Xinje XDPPro project, PLC1: XD5-60-6Pls (software 3.4 2016-10-12)

PROGRAM Ladder

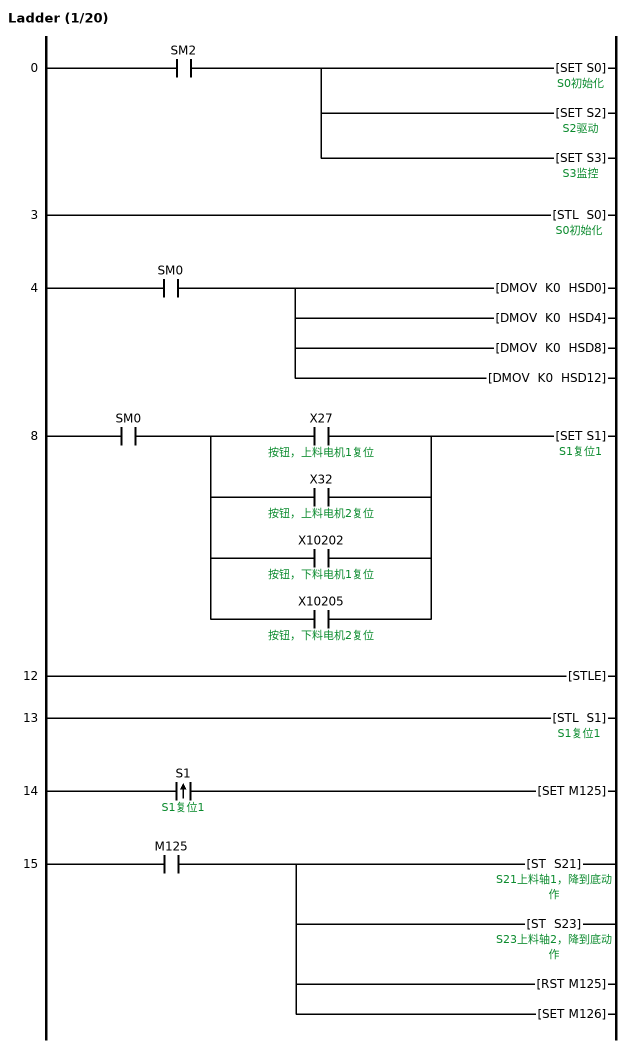
LD     SM2
SET    S0	; S0初始化
SET    S2	; S2驱动
SET    S3	; S3监控
STL    S0	; S0初始化
LD     SM0
DMOV   K0 HSD0
DMOV   K0 HSD4
DMOV   K0 HSD8
DMOV   K0 HSD12
LD     SM0
LD     X27	; 按钮，上料电机1复位
OR     X32	; 按钮，上料电机2复位
OR     X10202	; 按钮，下料电机1复位
OR     X10205	; 按钮，下料电机2复位
ANB
SET    S1	; S1复位1
STLE
STL    S1	; S1复位1
LDP    S1	; S1复位1
SET    M125
LD     M125
ST     S21	; S21上料轴1，降到底动作
ST     S23	; S23上料轴2，降到底动作
RST    M125
SET    M126

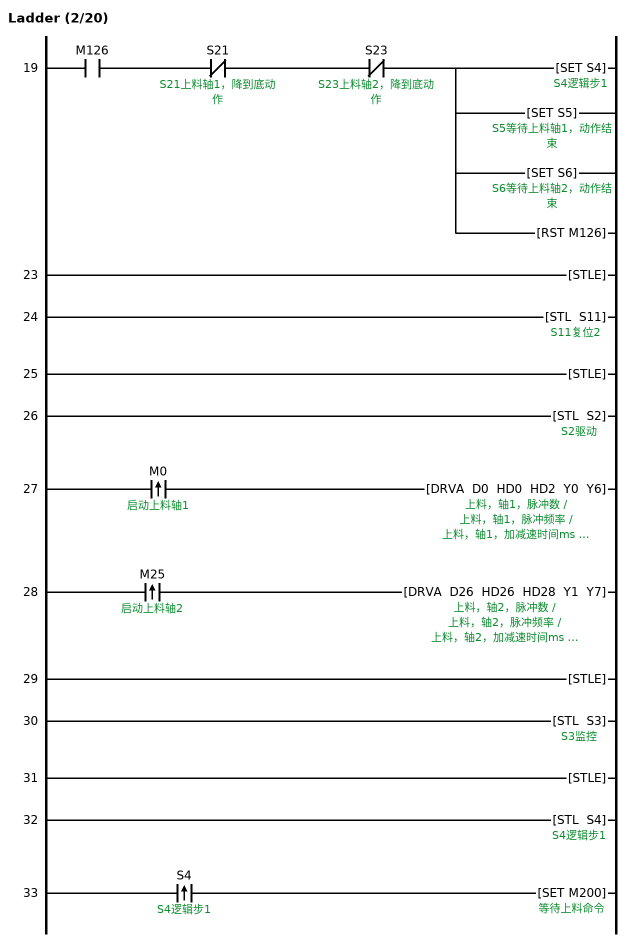
LD     M126
ANI    S21	; S21上料轴1，降到底动作
ANI    S23	; S23上料轴2，降到底动作
SET    S4	; S4逻辑步1
SET    S5	; S5等待上料轴1，动作结束
SET    S6	; S6等待上料轴2，动作结束
RST    M126
STLE
STL    S11	; S11复位2
STLE
STL    S2	; S2驱动
LDP    M0	; 启动上料轴1
DRVA   D0 HD0 HD2 Y0 Y6	; 上料，轴1，脉冲数 / 上料，轴1，脉冲频率 / 上料，轴1，加减速时间ms / 上料1电机脉冲 / 上料1电机方向
LDP    M25	; 启动上料轴2
DRVA   D26 HD26 HD28 Y1 Y7	; 上料，轴2，脉冲数 / 上料，轴2，脉冲频率 / 上料，轴2，加减速时间ms / 上料2电机脉冲 / 上料2电机方向
STLE
STL    S3	; S3监控
STLE
STL    S4	; S4逻辑步1
LDP    S4	; S4逻辑步1
SET    M200	; 等待上料命令

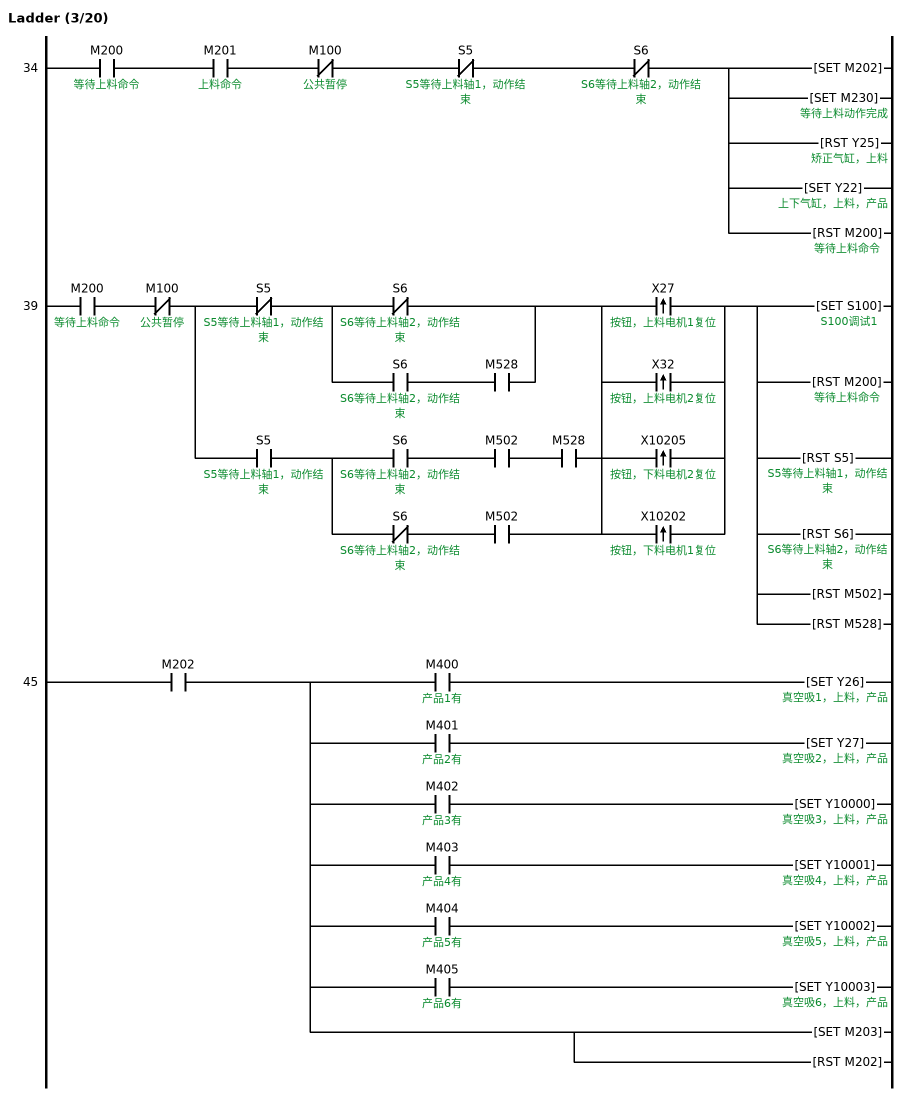
LD     M200	; 等待上料命令
AND    M201	; 上料命令
ANI    M100	; 公共暂停
ANI    S5	; S5等待上料轴1，动作结束
ANI    S6	; S6等待上料轴2，动作结束
SET    M202
SET    M230	; 等待上料动作完成
RST    Y25	; 矫正气缸，上料
SET    Y22	; 上下气缸，上料，产品
RST    M200	; 等待上料命令
LD     M200	; 等待上料命令
ANI    M100	; 公共暂停
LDI    S5	; S5等待上料轴1，动作结束
LDI    S6	; S6等待上料轴2，动作结束
LD     S6	; S6等待上料轴2，动作结束
AND    M528
ORB
ANB
LD     S5	; S5等待上料轴1，动作结束
LD     S6	; S6等待上料轴2，动作结束
AND    M502
AND    M528
LDI    S6	; S6等待上料轴2，动作结束
AND    M502
ORB
ANB
ORB
ANB
LDP    X27	; 按钮，上料电机1复位
ORP    X32	; 按钮，上料电机2复位
ORP    X10205	; 按钮，下料电机2复位
ORP    X10202	; 按钮，下料电机1复位
ANB
SET    S100	; S100调试1
RST    M200	; 等待上料命令
RST    S5	; S5等待上料轴1，动作结束
RST    S6	; S6等待上料轴2，动作结束
RST    M502
RST    M528
LD     M202
MPS
AND    M400	; 产品1有
SET    Y26	; 真空吸1，上料，产品
MRD
AND    M401	; 产品2有
SET    Y27	; 真空吸2，上料，产品
MRD
AND    M402	; 产品3有
SET    Y10000	; 真空吸3，上料，产品
MRD
AND    M403	; 产品4有
SET    Y10001	; 真空吸4，上料，产品
MRD
AND    M404	; 产品5有
SET    Y10002	; 真空吸5，上料，产品
MRD
AND    M405	; 产品6有
SET    Y10003	; 真空吸6，上料，产品
MPP
SET    M203
RST    M202

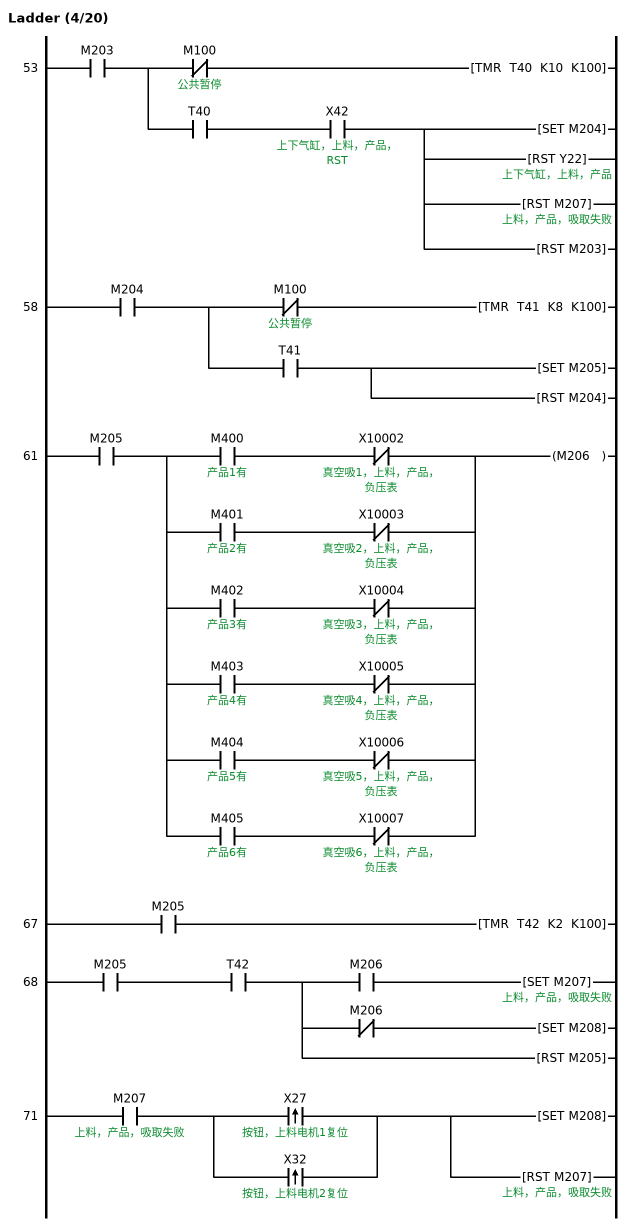
LD     M203
MPS
ANI    M100	; 公共暂停
TMR    T40 K10 K100
MPP
AND    T40
AND    X42	; 上下气缸，上料，产品，RST
SET    M204
RST    Y22	; 上下气缸，上料，产品
RST    M207	; 上料，产品，吸取失败
RST    M203
LD     M204
MPS
ANI    M100	; 公共暂停
TMR    T41 K8 K100
MPP
AND    T41
SET    M205
RST    M204
LD     M205
LD     M400	; 产品1有
ANI    X10002	; 真空吸1，上料，产品，负压表
LD     M401	; 产品2有
ANI    X10003	; 真空吸2，上料，产品，负压表
ORB
LD     M402	; 产品3有
ANI    X10004	; 真空吸3，上料，产品，负压表
ORB
LD     M403	; 产品4有
ANI    X10005	; 真空吸4，上料，产品，负压表
ORB
LD     M404	; 产品5有
ANI    X10006	; 真空吸5，上料，产品，负压表
ORB
LD     M405	; 产品6有
ANI    X10007	; 真空吸6，上料，产品，负压表
ORB
ANB
OUT    M206
LD     M205
TMR    T42 K2 K100
LD     M205
AND    T42
MPS
AND    M206
SET    M207	; 上料，产品，吸取失败
MRD
ANI    M206
SET    M208
MPP
RST    M205
LD     M207	; 上料，产品，吸取失败
LDP    X27	; 按钮，上料电机1复位
ORP    X32	; 按钮，上料电机2复位
ANB
SET    M208
RST    M207	; 上料，产品，吸取失败

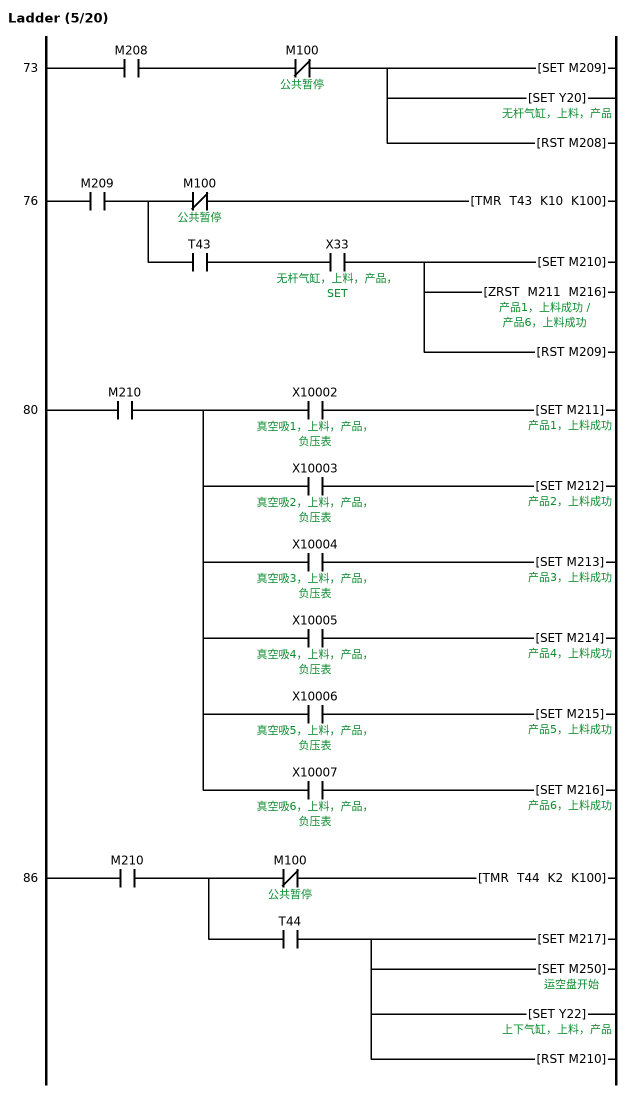
LD     M208
ANI    M100	; 公共暂停
SET    M209
SET    Y20	; 无杆气缸，上料，产品
RST    M208
LD     M209
MPS
ANI    M100	; 公共暂停
TMR    T43 K10 K100
MPP
AND    T43
AND    X33	; 无杆气缸，上料，产品，SET
SET    M210
ZRST   M211 M216	; 产品1，上料成功 / 产品6，上料成功
RST    M209
LD     M210
MPS
AND    X10002	; 真空吸1，上料，产品，负压表
SET    M211	; 产品1，上料成功
MRD
AND    X10003	; 真空吸2，上料，产品，负压表
SET    M212	; 产品2，上料成功
MRD
AND    X10004	; 真空吸3，上料，产品，负压表
SET    M213	; 产品3，上料成功
MRD
AND    X10005	; 真空吸4，上料，产品，负压表
SET    M214	; 产品4，上料成功
MRD
AND    X10006	; 真空吸5，上料，产品，负压表
SET    M215	; 产品5，上料成功
MPP
AND    X10007	; 真空吸6，上料，产品，负压表
SET    M216	; 产品6，上料成功
LD     M210
MPS
ANI    M100	; 公共暂停
TMR    T44 K2 K100
MPP
AND    T44
SET    M217
SET    M250	; 运空盘开始
SET    Y22	; 上下气缸，上料，产品
RST    M210

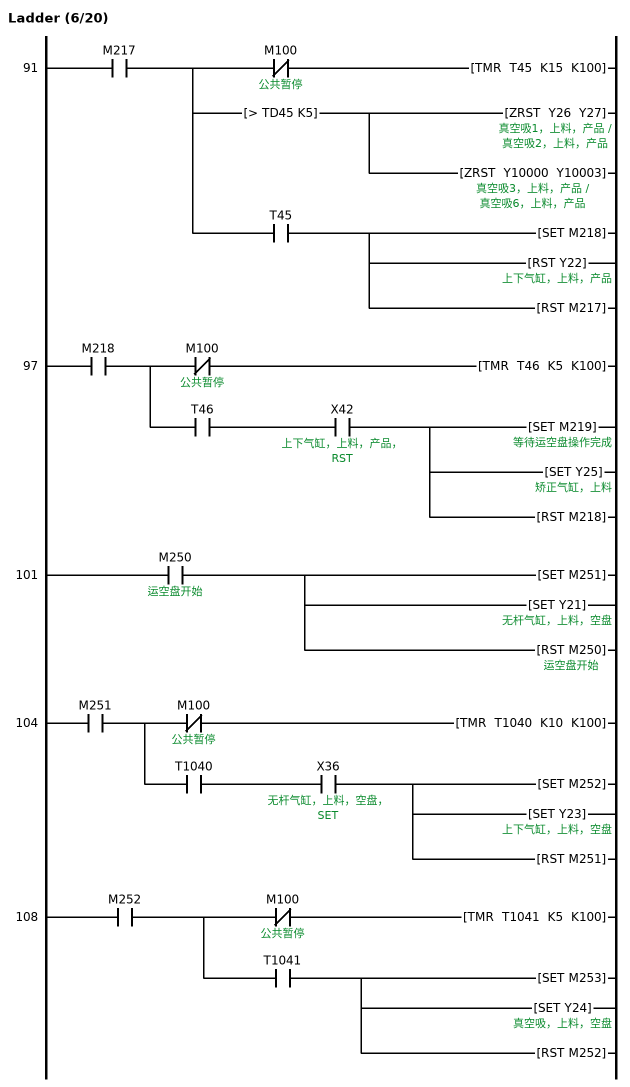
LD     M217
MPS
ANI    M100	; 公共暂停
TMR    T45 K15 K100
MRD
AND>   TD45 K5
ZRST   Y26 Y27	; 真空吸1，上料，产品 / 真空吸2，上料，产品
ZRST   Y10000 Y10003	; 真空吸3，上料，产品 / 真空吸6，上料，产品
MPP
AND    T45
SET    M218
RST    Y22	; 上下气缸，上料，产品
RST    M217
LD     M218
MPS
ANI    M100	; 公共暂停
TMR    T46 K5 K100
MPP
AND    T46
AND    X42	; 上下气缸，上料，产品，RST
SET    M219	; 等待运空盘操作完成
SET    Y25	; 矫正气缸，上料
RST    M218
LD     M250	; 运空盘开始
SET    M251
SET    Y21	; 无杆气缸，上料，空盘
RST    M250	; 运空盘开始
LD     M251
MPS
ANI    M100	; 公共暂停
TMR    T1040 K10 K100
MPP
AND    T1040
AND    X36	; 无杆气缸，上料，空盘，SET
SET    M252
SET    Y23	; 上下气缸，上料，空盘
RST    M251
LD     M252
MPS
ANI    M100	; 公共暂停
TMR    T1041 K5 K100
MPP
AND    T1041
SET    M253
SET    Y24	; 真空吸，上料，空盘
RST    M252

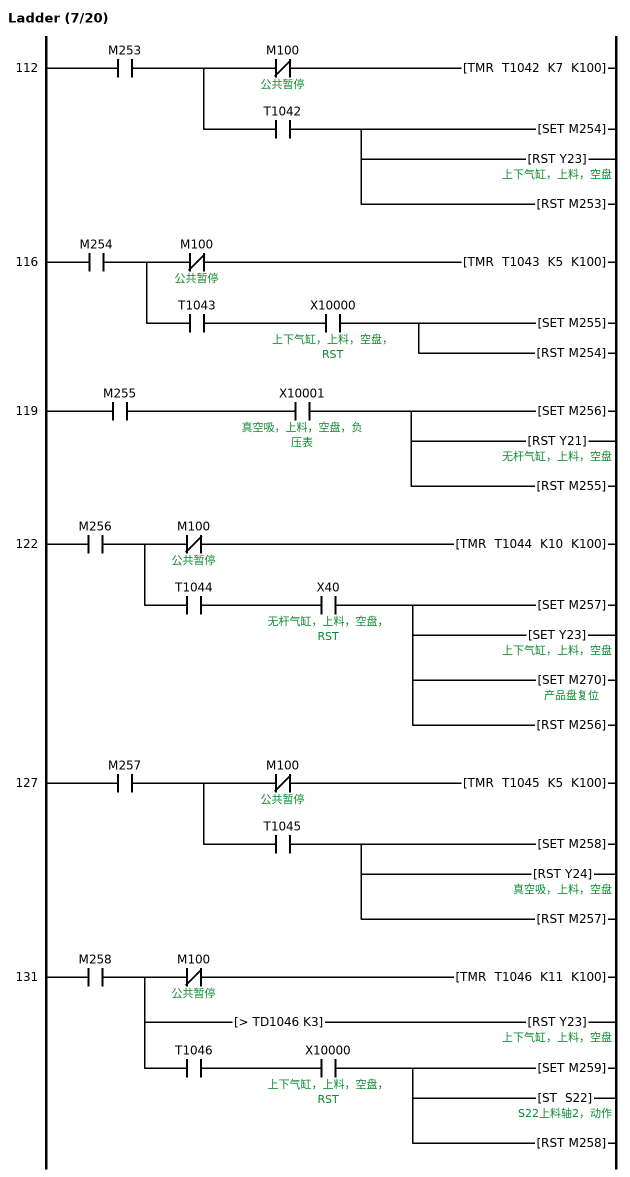
LD     M253
MPS
ANI    M100	; 公共暂停
TMR    T1042 K7 K100
MPP
AND    T1042
SET    M254
RST    Y23	; 上下气缸，上料，空盘
RST    M253
LD     M254
MPS
ANI    M100	; 公共暂停
TMR    T1043 K5 K100
MPP
AND    T1043
AND    X10000	; 上下气缸，上料，空盘，RST
SET    M255
RST    M254
LD     M255
AND    X10001	; 真空吸，上料，空盘，负压表
SET    M256
RST    Y21	; 无杆气缸，上料，空盘
RST    M255
LD     M256
MPS
ANI    M100	; 公共暂停
TMR    T1044 K10 K100
MPP
AND    T1044
AND    X40	; 无杆气缸，上料，空盘，RST
SET    M257
SET    Y23	; 上下气缸，上料，空盘
SET    M270	; 产品盘复位
RST    M256
LD     M257
MPS
ANI    M100	; 公共暂停
TMR    T1045 K5 K100
MPP
AND    T1045
SET    M258
RST    Y24	; 真空吸，上料，空盘
RST    M257
LD     M258
MPS
ANI    M100	; 公共暂停
TMR    T1046 K11 K100
MRD
AND>   TD1046 K3
RST    Y23	; 上下气缸，上料，空盘
MPP
AND    T1046
AND    X10000	; 上下气缸，上料，空盘，RST
SET    M259
ST     S22	; S22上料轴2，动作
RST    M258

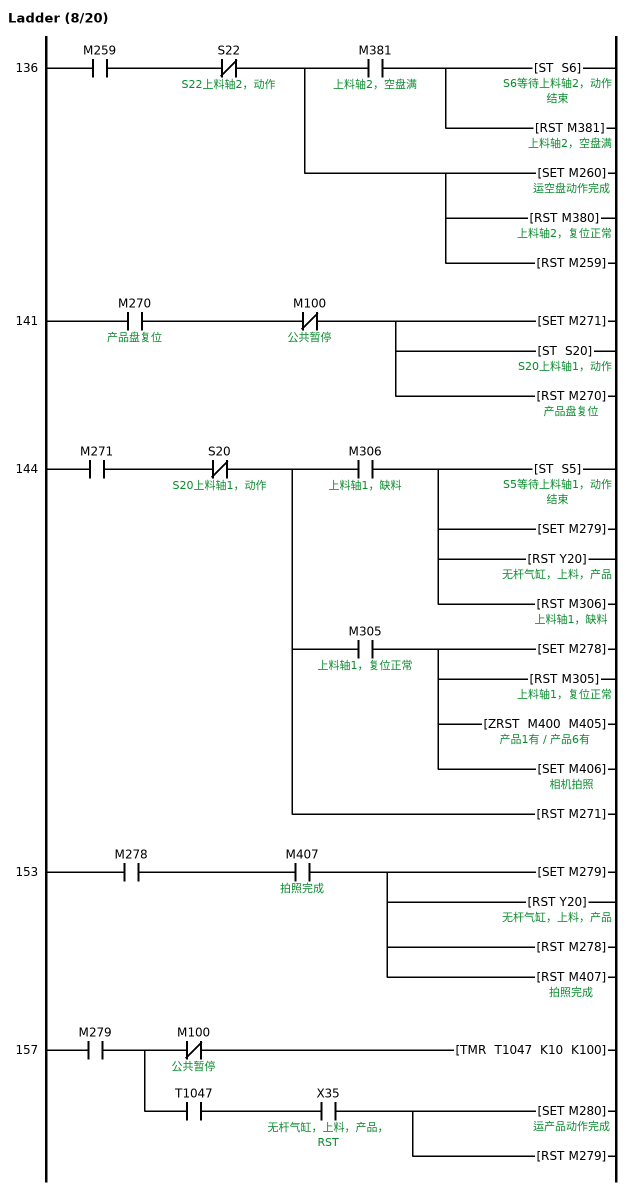
LD     M259
ANI    S22	; S22上料轴2，动作
MPS
AND    M381	; 上料轴2，空盘满
ST     S6	; S6等待上料轴2，动作结束
RST    M381	; 上料轴2，空盘满
MPP
SET    M260	; 运空盘动作完成
RST    M380	; 上料轴2，复位正常
RST    M259
LD     M270	; 产品盘复位
ANI    M100	; 公共暂停
SET    M271
ST     S20	; S20上料轴1，动作
RST    M270	; 产品盘复位
LD     M271
ANI    S20	; S20上料轴1，动作
MPS
AND    M306	; 上料轴1，缺料
ST     S5	; S5等待上料轴1，动作结束
SET    M279
RST    Y20	; 无杆气缸，上料，产品
RST    M306	; 上料轴1，缺料
MRD
AND    M305	; 上料轴1，复位正常
SET    M278
RST    M305	; 上料轴1，复位正常
ZRST   M400 M405	; 产品1有 / 产品6有
SET    M406	; 相机拍照
MPP
RST    M271
LD     M278
AND    M407	; 拍照完成
SET    M279
RST    Y20	; 无杆气缸，上料，产品
RST    M278
RST    M407	; 拍照完成
LD     M279
MPS
ANI    M100	; 公共暂停
TMR    T1047 K10 K100
MPP
AND    T1047
AND    X35	; 无杆气缸，上料，产品，RST
SET    M280	; 运产品动作完成
RST    M279

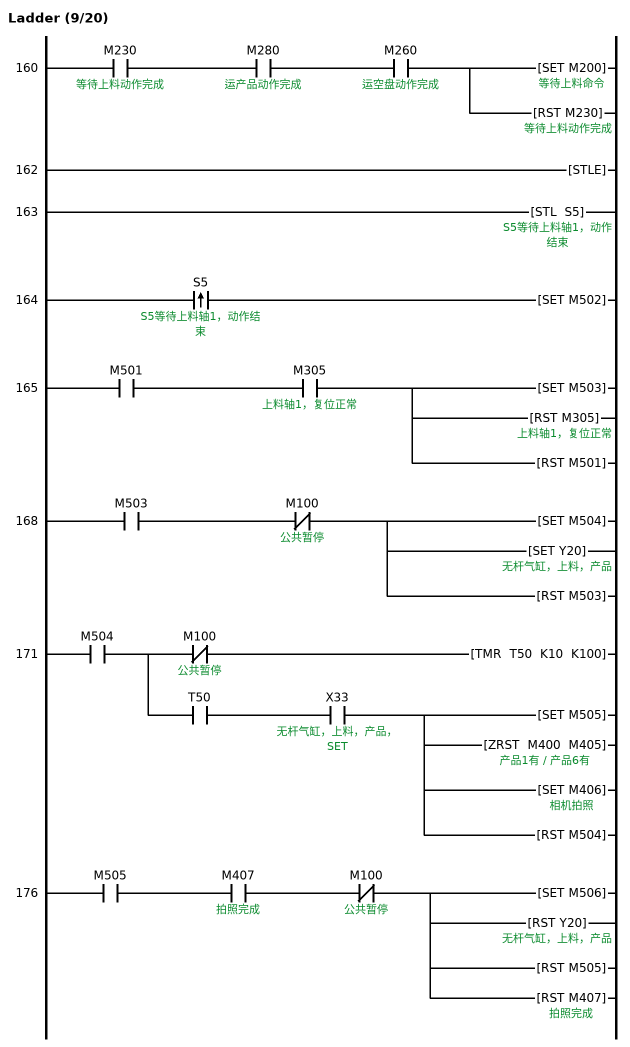
LD     M230	; 等待上料动作完成
AND    M280	; 运产品动作完成
AND    M260	; 运空盘动作完成
SET    M200	; 等待上料命令
RST    M230	; 等待上料动作完成
STLE
STL    S5	; S5等待上料轴1，动作结束
LDP    S5	; S5等待上料轴1，动作结束
SET    M502
LD     M501
AND    M305	; 上料轴1，复位正常
SET    M503
RST    M305	; 上料轴1，复位正常
RST    M501
LD     M503
ANI    M100	; 公共暂停
SET    M504
SET    Y20	; 无杆气缸，上料，产品
RST    M503
LD     M504
MPS
ANI    M100	; 公共暂停
TMR    T50 K10 K100
MPP
AND    T50
AND    X33	; 无杆气缸，上料，产品，SET
SET    M505
ZRST   M400 M405	; 产品1有 / 产品6有
SET    M406	; 相机拍照
RST    M504
LD     M505
AND    M407	; 拍照完成
ANI    M100	; 公共暂停
SET    M506
RST    Y20	; 无杆气缸，上料，产品
RST    M505
RST    M407	; 拍照完成

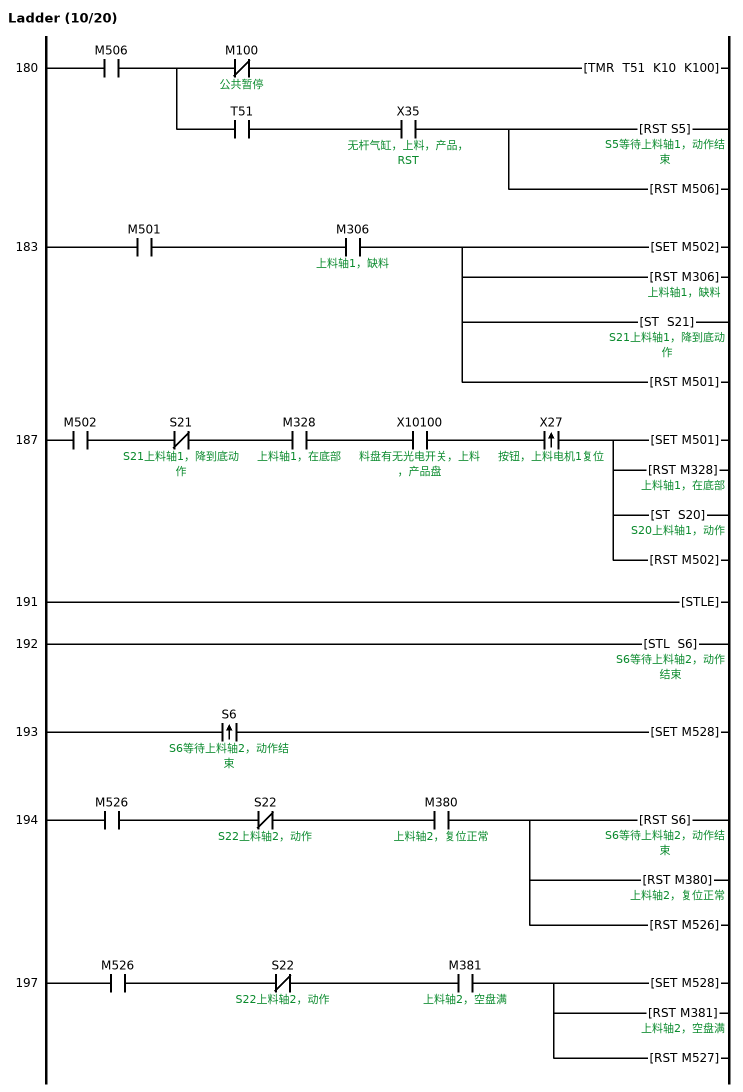
LD     M506
MPS
ANI    M100	; 公共暂停
TMR    T51 K10 K100
MPP
AND    T51
AND    X35	; 无杆气缸，上料，产品，RST
RST    S5	; S5等待上料轴1，动作结束
RST    M506
LD     M501
AND    M306	; 上料轴1，缺料
SET    M502
RST    M306	; 上料轴1，缺料
ST     S21	; S21上料轴1，降到底动作
RST    M501
LD     M502
ANI    S21	; S21上料轴1，降到底动作
AND    M328	; 上料轴1，在底部
AND    X10100	; 料盘有无光电开关，上料，产品盘
ANDP   X27	; 按钮，上料电机1复位
SET    M501
RST    M328	; 上料轴1，在底部
ST     S20	; S20上料轴1，动作
RST    M502
STLE
STL    S6	; S6等待上料轴2，动作结束
LDP    S6	; S6等待上料轴2，动作结束
SET    M528
LD     M526
ANI    S22	; S22上料轴2，动作
AND    M380	; 上料轴2，复位正常
RST    S6	; S6等待上料轴2，动作结束
RST    M380	; 上料轴2，复位正常
RST    M526
LD     M526
ANI    S22	; S22上料轴2，动作
AND    M381	; 上料轴2，空盘满
SET    M528
RST    M381	; 上料轴2，空盘满
RST    M527

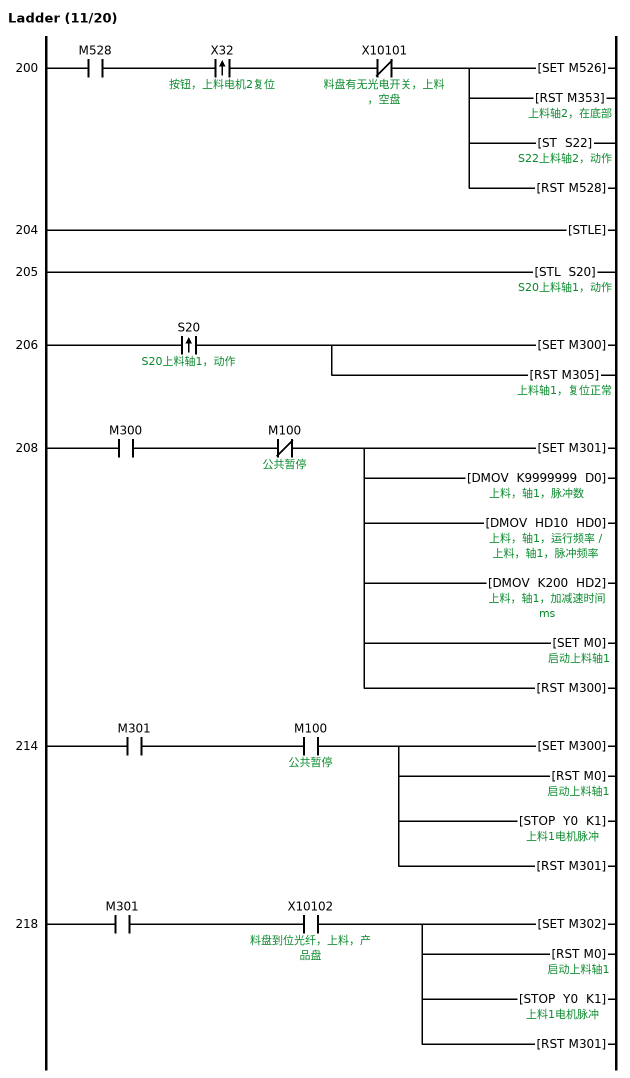
LD     M528
ANDP   X32	; 按钮，上料电机2复位
ANI    X10101	; 料盘有无光电开关，上料，空盘
SET    M526
RST    M353	; 上料轴2，在底部
ST     S22	; S22上料轴2，动作
RST    M528
STLE
STL    S20	; S20上料轴1，动作
LDP    S20	; S20上料轴1，动作
SET    M300
RST    M305	; 上料轴1，复位正常
LD     M300
ANI    M100	; 公共暂停
SET    M301
DMOV   K9999999 D0	; 上料，轴1，脉冲数
DMOV   HD10 HD0	; 上料，轴1，运行频率 / 上料，轴1，脉冲频率
DMOV   K200 HD2	; 上料，轴1，加减速时间ms
SET    M0	; 启动上料轴1
RST    M300
LD     M301
AND    M100	; 公共暂停
SET    M300
RST    M0	; 启动上料轴1
STOP   Y0 K1	; 上料1电机脉冲
RST    M301
LD     M301
AND    X10102	; 料盘到位光纤，上料，产品盘
SET    M302
RST    M0	; 启动上料轴1
STOP   Y0 K1	; 上料1电机脉冲
RST    M301

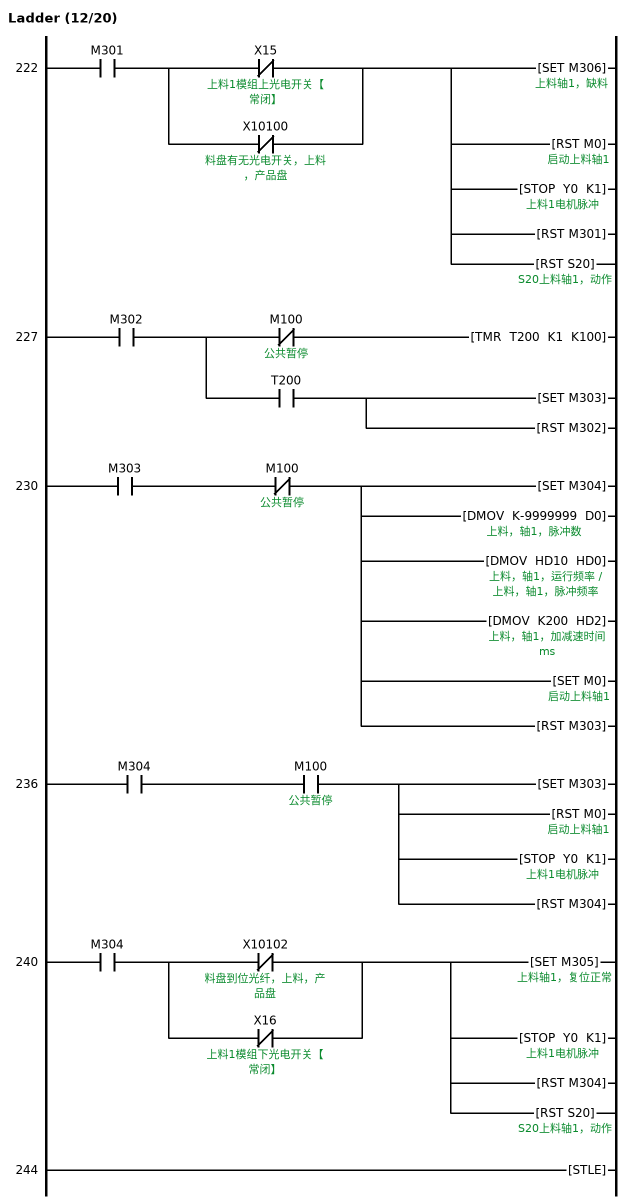
LD     M301
LDI    X15	; 上料1模组上光电开关【常闭】
ORI    X10100	; 料盘有无光电开关，上料，产品盘
ANB
SET    M306	; 上料轴1，缺料
RST    M0	; 启动上料轴1
STOP   Y0 K1	; 上料1电机脉冲
RST    M301
RST    S20	; S20上料轴1，动作
LD     M302
MPS
ANI    M100	; 公共暂停
TMR    T200 K1 K100
MPP
AND    T200
SET    M303
RST    M302
LD     M303
ANI    M100	; 公共暂停
SET    M304
DMOV   K-9999999 D0	; 上料，轴1，脉冲数
DMOV   HD10 HD0	; 上料，轴1，运行频率 / 上料，轴1，脉冲频率
DMOV   K200 HD2	; 上料，轴1，加减速时间ms
SET    M0	; 启动上料轴1
RST    M303
LD     M304
AND    M100	; 公共暂停
SET    M303
RST    M0	; 启动上料轴1
STOP   Y0 K1	; 上料1电机脉冲
RST    M304
LD     M304
LDI    X10102	; 料盘到位光纤，上料，产品盘
ORI    X16	; 上料1模组下光电开关【常闭】
ANB
SET    M305	; 上料轴1，复位正常
STOP   Y0 K1	; 上料1电机脉冲
RST    M304
RST    S20	; S20上料轴1，动作
STLE

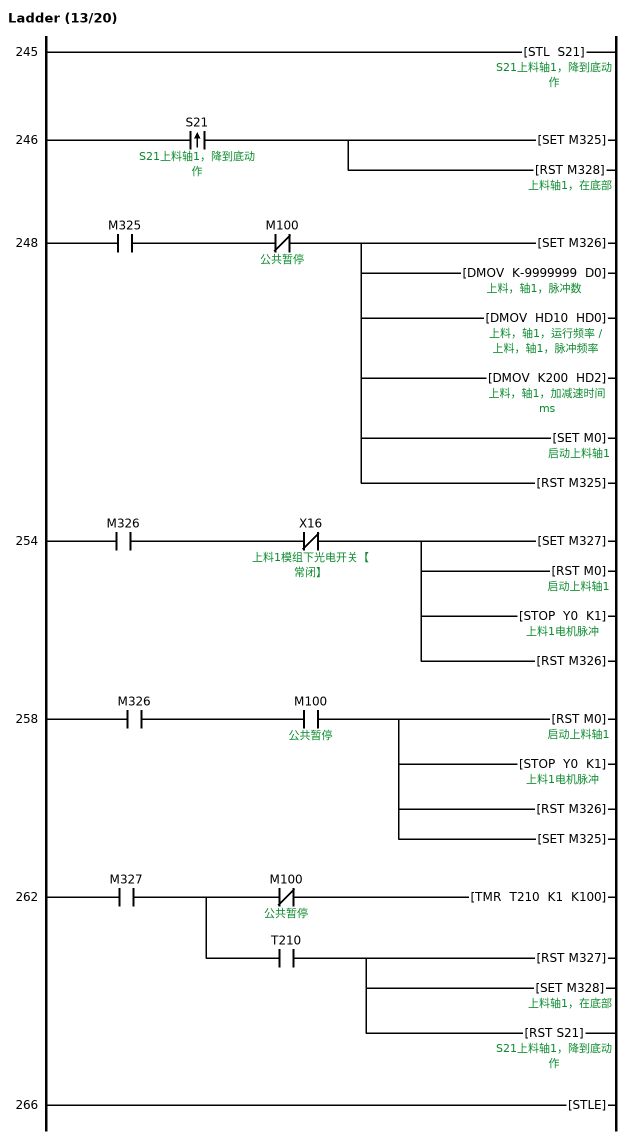
STL    S21	; S21上料轴1，降到底动作
LDP    S21	; S21上料轴1，降到底动作
SET    M325
RST    M328	; 上料轴1，在底部
LD     M325
ANI    M100	; 公共暂停
SET    M326
DMOV   K-9999999 D0	; 上料，轴1，脉冲数
DMOV   HD10 HD0	; 上料，轴1，运行频率 / 上料，轴1，脉冲频率
DMOV   K200 HD2	; 上料，轴1，加减速时间ms
SET    M0	; 启动上料轴1
RST    M325
LD     M326
ANI    X16	; 上料1模组下光电开关【常闭】
SET    M327
RST    M0	; 启动上料轴1
STOP   Y0 K1	; 上料1电机脉冲
RST    M326
LD     M326
AND    M100	; 公共暂停
RST    M0	; 启动上料轴1
STOP   Y0 K1	; 上料1电机脉冲
RST    M326
SET    M325
LD     M327
MPS
ANI    M100	; 公共暂停
TMR    T210 K1 K100
MPP
AND    T210
RST    M327
SET    M328	; 上料轴1，在底部
RST    S21	; S21上料轴1，降到底动作
STLE

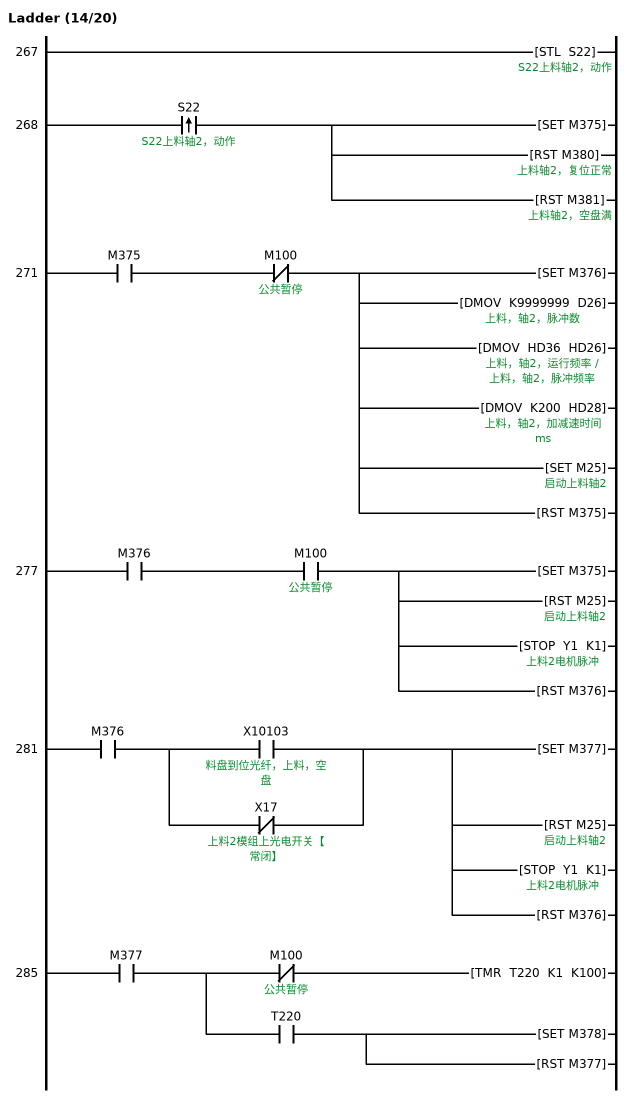
STL    S22	; S22上料轴2，动作
LDP    S22	; S22上料轴2，动作
SET    M375
RST    M380	; 上料轴2，复位正常
RST    M381	; 上料轴2，空盘满
LD     M375
ANI    M100	; 公共暂停
SET    M376
DMOV   K9999999 D26	; 上料，轴2，脉冲数
DMOV   HD36 HD26	; 上料，轴2，运行频率 / 上料，轴2，脉冲频率
DMOV   K200 HD28	; 上料，轴2，加减速时间ms
SET    M25	; 启动上料轴2
RST    M375
LD     M376
AND    M100	; 公共暂停
SET    M375
RST    M25	; 启动上料轴2
STOP   Y1 K1	; 上料2电机脉冲
RST    M376
LD     M376
LD     X10103	; 料盘到位光纤，上料，空盘
ORI    X17	; 上料2模组上光电开关【常闭】
ANB
SET    M377
RST    M25	; 启动上料轴2
STOP   Y1 K1	; 上料2电机脉冲
RST    M376
LD     M377
MPS
ANI    M100	; 公共暂停
TMR    T220 K1 K100
MPP
AND    T220
SET    M378
RST    M377

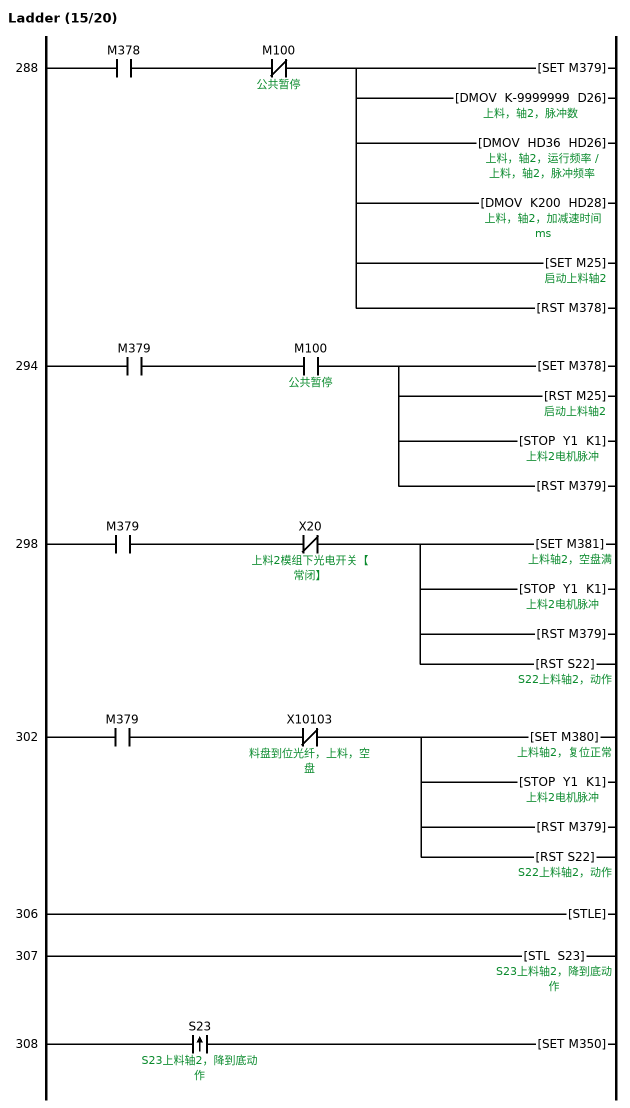
LD     M378
ANI    M100	; 公共暂停
SET    M379
DMOV   K-9999999 D26	; 上料，轴2，脉冲数
DMOV   HD36 HD26	; 上料，轴2，运行频率 / 上料，轴2，脉冲频率
DMOV   K200 HD28	; 上料，轴2，加减速时间ms
SET    M25	; 启动上料轴2
RST    M378
LD     M379
AND    M100	; 公共暂停
SET    M378
RST    M25	; 启动上料轴2
STOP   Y1 K1	; 上料2电机脉冲
RST    M379
LD     M379
ANI    X20	; 上料2模组下光电开关【常闭】
SET    M381	; 上料轴2，空盘满
STOP   Y1 K1	; 上料2电机脉冲
RST    M379
RST    S22	; S22上料轴2，动作
LD     M379
ANI    X10103	; 料盘到位光纤，上料，空盘
SET    M380	; 上料轴2，复位正常
STOP   Y1 K1	; 上料2电机脉冲
RST    M379
RST    S22	; S22上料轴2，动作
STLE
STL    S23	; S23上料轴2，降到底动作
LDP    S23	; S23上料轴2，降到底动作
SET    M350

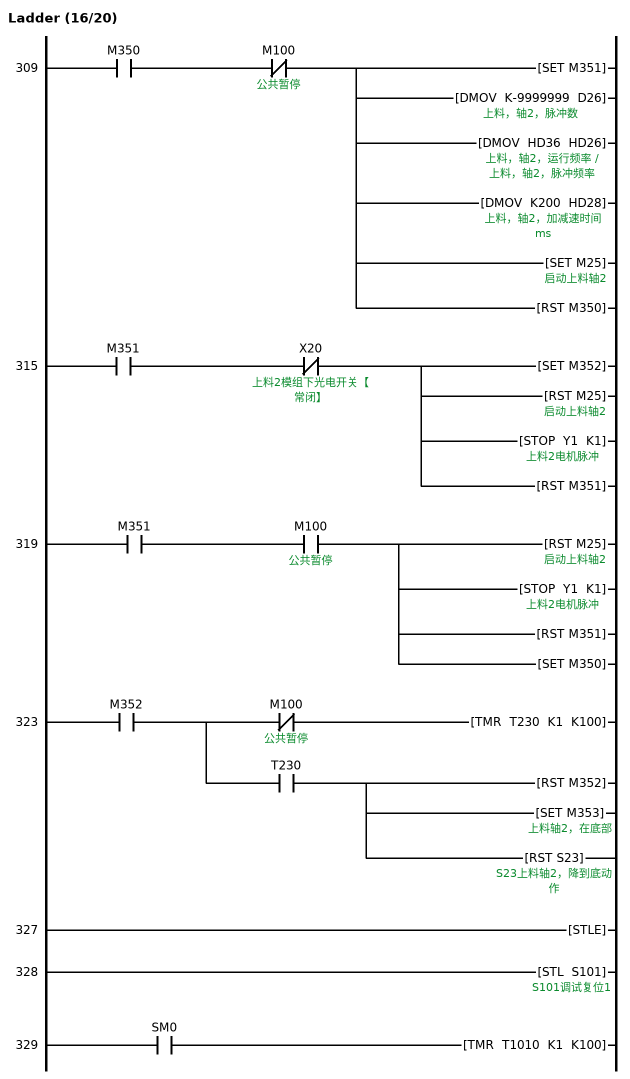
LD     M350
ANI    M100	; 公共暂停
SET    M351
DMOV   K-9999999 D26	; 上料，轴2，脉冲数
DMOV   HD36 HD26	; 上料，轴2，运行频率 / 上料，轴2，脉冲频率
DMOV   K200 HD28	; 上料，轴2，加减速时间ms
SET    M25	; 启动上料轴2
RST    M350
LD     M351
ANI    X20	; 上料2模组下光电开关【常闭】
SET    M352
RST    M25	; 启动上料轴2
STOP   Y1 K1	; 上料2电机脉冲
RST    M351
LD     M351
AND    M100	; 公共暂停
RST    M25	; 启动上料轴2
STOP   Y1 K1	; 上料2电机脉冲
RST    M351
SET    M350
LD     M352
MPS
ANI    M100	; 公共暂停
TMR    T230 K1 K100
MPP
AND    T230
RST    M352
SET    M353	; 上料轴2，在底部
RST    S23	; S23上料轴2，降到底动作
STLE
STL    S101	; S101调试复位1
LD     SM0
TMR    T1010 K1 K100

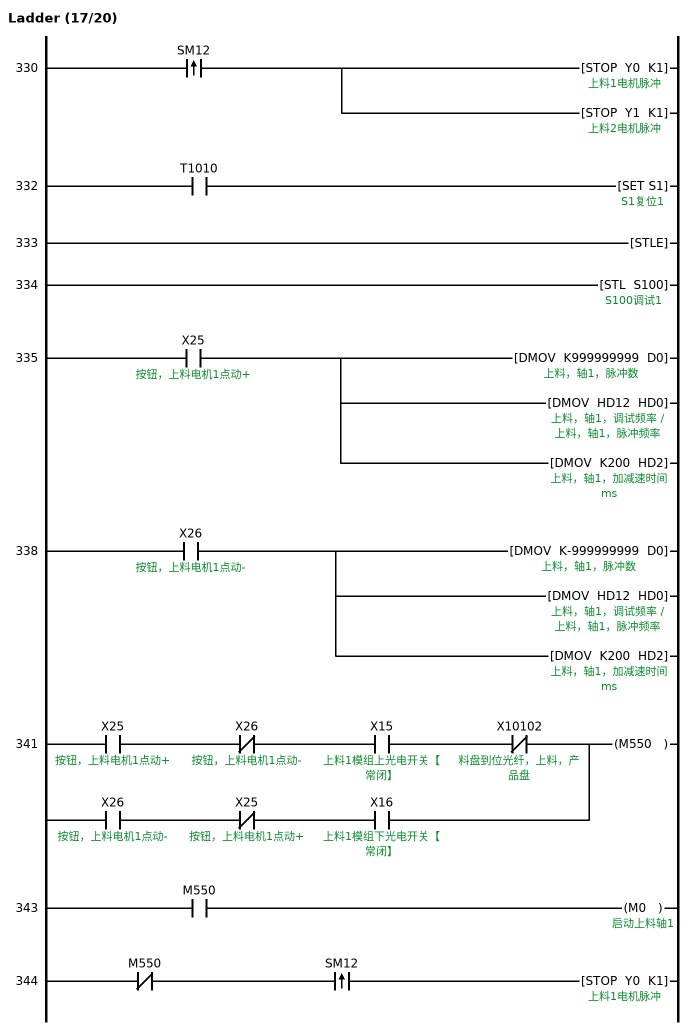
LDP    SM12
STOP   Y0 K1	; 上料1电机脉冲
STOP   Y1 K1	; 上料2电机脉冲
LD     T1010
SET    S1	; S1复位1
STLE
STL    S100	; S100调试1
LD     X25	; 按钮，上料电机1点动+
DMOV   K999999999 D0	; 上料，轴1，脉冲数
DMOV   HD12 HD0	; 上料，轴1，调试频率 / 上料，轴1，脉冲频率
DMOV   K200 HD2	; 上料，轴1，加减速时间ms
LD     X26	; 按钮，上料电机1点动-
DMOV   K-999999999 D0	; 上料，轴1，脉冲数
DMOV   HD12 HD0	; 上料，轴1，调试频率 / 上料，轴1，脉冲频率
DMOV   K200 HD2	; 上料，轴1，加减速时间ms
LD     X25	; 按钮，上料电机1点动+
ANI    X26	; 按钮，上料电机1点动-
AND    X15	; 上料1模组上光电开关【常闭】
ANI    X10102	; 料盘到位光纤，上料，产品盘
LD     X26	; 按钮，上料电机1点动-
ANI    X25	; 按钮，上料电机1点动+
AND    X16	; 上料1模组下光电开关【常闭】
ORB
OUT    M550
LD     M550
OUT    M0	; 启动上料轴1
LDI    M550
ANDP   SM12
STOP   Y0 K1	; 上料1电机脉冲

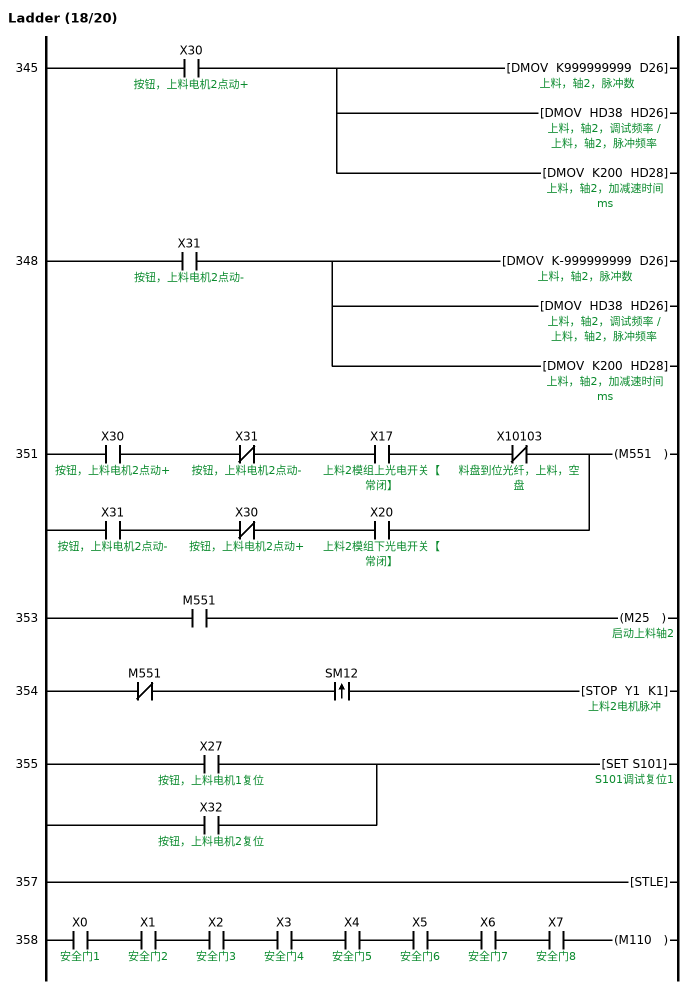
LD     X30	; 按钮，上料电机2点动+
DMOV   K999999999 D26	; 上料，轴2，脉冲数
DMOV   HD38 HD26	; 上料，轴2，调试频率 / 上料，轴2，脉冲频率
DMOV   K200 HD28	; 上料，轴2，加减速时间ms
LD     X31	; 按钮，上料电机2点动-
DMOV   K-999999999 D26	; 上料，轴2，脉冲数
DMOV   HD38 HD26	; 上料，轴2，调试频率 / 上料，轴2，脉冲频率
DMOV   K200 HD28	; 上料，轴2，加减速时间ms
LD     X30	; 按钮，上料电机2点动+
ANI    X31	; 按钮，上料电机2点动-
AND    X17	; 上料2模组上光电开关【常闭】
ANI    X10103	; 料盘到位光纤，上料，空盘
LD     X31	; 按钮，上料电机2点动-
ANI    X30	; 按钮，上料电机2点动+
AND    X20	; 上料2模组下光电开关【常闭】
ORB
OUT    M551
LD     M551
OUT    M25	; 启动上料轴2
LDI    M551
ANDP   SM12
STOP   Y1 K1	; 上料2电机脉冲
LD     X27	; 按钮，上料电机1复位
OR     X32	; 按钮，上料电机2复位
SET    S101	; S101调试复位1
STLE
LD     X0	; 安全门1
AND    X1	; 安全门2
AND    X2	; 安全门3
AND    X3	; 安全门4
AND    X4	; 安全门5
AND    X5	; 安全门6
AND    X6	; 安全门7
AND    X7	; 安全门8
OUT    M110

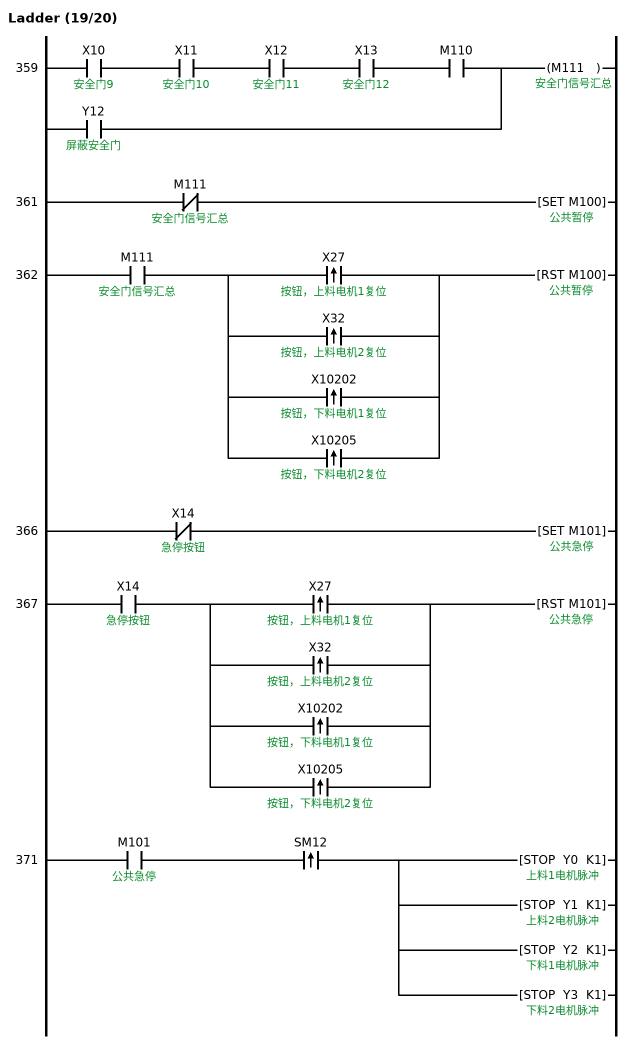
LD     X10	; 安全门9
AND    X11	; 安全门10
AND    X12	; 安全门11
AND    X13	; 安全门12
AND    M110
OR     Y12	; 屏蔽安全门
OUT    M111	; 安全门信号汇总
LDI    M111	; 安全门信号汇总
SET    M100	; 公共暂停
LD     M111	; 安全门信号汇总
LDP    X27	; 按钮，上料电机1复位
ORP    X32	; 按钮，上料电机2复位
ORP    X10202	; 按钮，下料电机1复位
ORP    X10205	; 按钮，下料电机2复位
ANB
RST    M100	; 公共暂停
LDI    X14	; 急停按钮
SET    M101	; 公共急停
LD     X14	; 急停按钮
LDP    X27	; 按钮，上料电机1复位
ORP    X32	; 按钮，上料电机2复位
ORP    X10202	; 按钮，下料电机1复位
ORP    X10205	; 按钮，下料电机2复位
ANB
RST    M101	; 公共急停
LD     M101	; 公共急停
ANDP   SM12
STOP   Y0 K1	; 上料1电机脉冲
STOP   Y1 K1	; 上料2电机脉冲
STOP   Y2 K1	; 下料1电机脉冲
STOP   Y3 K1	; 下料2电机脉冲

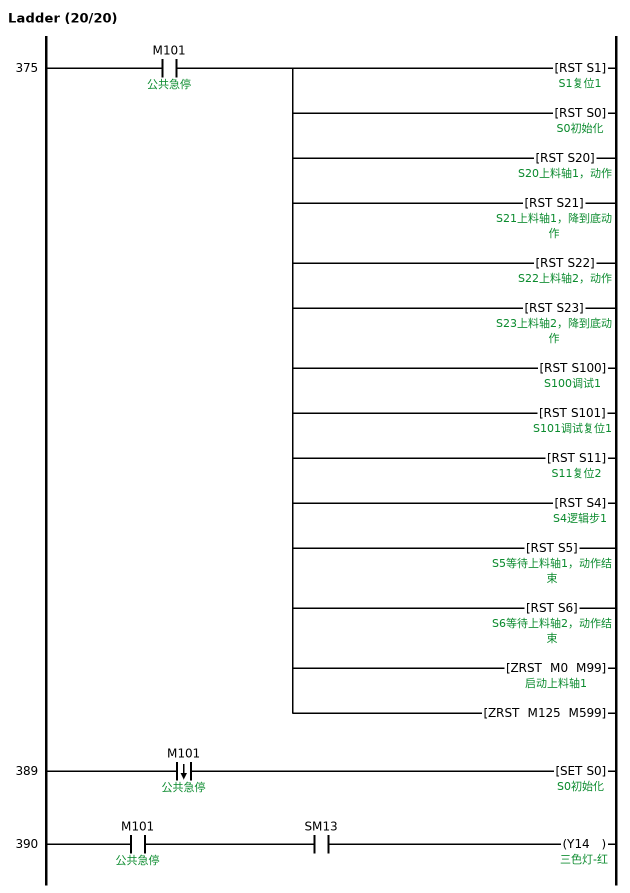
LD     M101	; 公共急停
RST    S1	; S1复位1
RST    S0	; S0初始化
RST    S20	; S20上料轴1，动作
RST    S21	; S21上料轴1，降到底动作
RST    S22	; S22上料轴2，动作
RST    S23	; S23上料轴2，降到底动作
RST    S100	; S100调试1
RST    S101	; S101调试复位1
RST    S11	; S11复位2
RST    S4	; S4逻辑步1
RST    S5	; S5等待上料轴1，动作结束
RST    S6	; S6等待上料轴2，动作结束
ZRST   M0 M99	; 启动上料轴1
ZRST   M125 M599
LDF    M101	; 公共急停
SET    S0	; S0初始化
LD     M101	; 公共急停
AND    SM13
OUT    Y14	; 三色灯-红

COMMENTS (devices not used above)
X21	下料1模组上光电开关【常闭】
X22	下料1模组下光电开关【常闭】
X23	下料2模组上光电开关【常闭】
X24	下料2模组下光电开关【常闭】
X41	上下气缸，上料，产品，SET
X43	上下气缸，上料，空盘，SET
X10104	无杆气缸，下料，空盘，SET
X10105	无杆气缸，下料，空盘，MID
X10106	无杆气缸，下料，空盘，RST
X10107	上下气缸，下料，空盘，SET
X10110	上下气缸，下料，空盘，RST
X10111	真空吸，下料，空盘，负压表
X10112	料盘有无光电开关，下料，产品盘
X10113	料盘有无光电开关，下料，空盘
X10114	料盘到位光纤，下料，产品盘
X10115	料盘到位光纤，下料，空盘
X10200	按钮，下料电机1点动+
X10201	按钮，下料电机1点动-
X10203	按钮，下料电机2点动+
X10204	按钮，下料电机2点动-
Y10	下料1电机方向
Y11	下料2电机方向
Y13	电磁铁
Y15	三色灯-黄
Y16	三色灯-绿
Y17	三色灯-蜂鸣器
Y10004	无杆气缸，下料，空盘
Y10005	上下气缸，下料，空盘
Y10006	真空吸，下料，空盘
M175	上料轴1，准备好
M176	上料轴2，准备好
M177	上料轴1，新上料
M243	报警：上料，缺料
M261	报警：空盘满，需要取走空盘
M272	报警：上料缺料
S30	S30上料，运产品，动作
T0	上料，轴1，上到位延时